(* CODESYS project FU_sDeleteRightBI.xml

Project tree, tasks and I/O mapping:
  function FU_sDeleteRightBI [ST]
*)

// FU_sDeleteRightBI
//This functions deletes a part of a string values are counted from the right instead of the left
// +-----------+----------+----------+-----------------------------------------------------------------------------------------------------------------------+
// |**Version**|**Author**| **Date** |**Changes**                                                                                                            |
// +-----------+----------+----------+-----------------------------------------------------------------------------------------------------------------------+
// | 1         | NSN      | 22-02-19 | Creation                                                                                                              |
// +-----------+----------+----------+-----------------------------------------------------------------------------------------------------------------------+
FUNCTION FU_sDeleteRightBI : STRING(255)
VAR_IN_OUT
	sStr		:STRING(1);			//Input String	
END_VAR
VAR_INPUT
	wLen		:WORD;				//Amount to trim from end
	wPos		:WORD;				//Position to delete from
END_VAR

FU_sDeleteRightBIBO(sOut:= FU_sDeleteRightBI, sStr:= sStr, wLen:= wLen,wPos:= wPos, wOutSize:= 255);

END_FUNCTION
